(* PLC project Beremiz Modbus Study PLC, Study Stand Beremiz Study PLC 1 *)
(* stored: creationDateTime 2026-06-11T14:12:07, modificationDateTime 2026-06-11T15:00:00 *)

PROGRAM plc_prg
  VAR
    ReadRequestExecute AT %QX0.0.0.0.0 : BOOL;
    WriteRequestExecute AT %QX0.0.1.0.0 : BOOL;
  END_VAR
  VAR
    SensorRegister AT %IW0.0.0.0 : WORD;
    RemoteOutputRegister AT %IW0.0.0.1 : WORD;
    ThresholdRegister AT %IW0.0.0.2 : WORD;
    OutputCommandRegister AT %QW0.0.1.1 : WORD;
  END_VAR
  VAR
    sensor_value : UINT;
    threshold : UINT;
    remote_output_echo : UINT;
    alarm : BOOL;
    output_command : UINT;
  END_VAR

            ReadRequestExecute := TRUE;
WriteRequestExecute := TRUE;

sensor_value := WORD_TO_UINT(SensorRegister);
threshold := WORD_TO_UINT(ThresholdRegister);
remote_output_echo := WORD_TO_UINT(RemoteOutputRegister);

alarm := sensor_value > threshold;

IF alarm THEN
    output_command := UINT#1;
ELSE
    output_command := UINT#0;
END_IF;

OutputCommandRegister := UINT_TO_WORD(output_command);
          
END_PROGRAM

CONFIGURATION config
  RESOURCE resource1 ON PLC
    TASK task0(INTERVAL := T#100ms, PRIORITY := 0);
    PROGRAM instance0 WITH task0 : plc_prg;
  END_RESOURCE
END_CONFIGURATION
